// TIA Portal V20 export
FUNCTION_BLOCK "SysPos"   // FB2010, FBD
TITLE = manage a standard positioning system
{ S7_Optimized_Access := 'TRUE' }
AUTHOR : MiCROTEC
VERSION : 1.2
// -2017.03 : Martin
// stored: AutoNumber false, MemoryReserve 100, SetENOAutomatically false
   VAR_INPUT
      actual { ExternalAccessible := 'False'; ExternalVisible := 'False'; ExternalWritable := 'False'} : Real;   // actual position
      target { ExternalAccessible := 'False'; ExternalVisible := 'False'; ExternalWritable := 'False'} : Real;   // target position , start new position only if target position change
      tarMinPos { ExternalAccessible := 'False'; ExternalVisible := 'False'; ExternalWritable := 'False'} : Real;   // target position minimum
      tarMaxPos { ExternalAccessible := 'False'; ExternalVisible := 'False'; ExternalWritable := 'False'} : Real;   // target position maximum
      tolerance { ExternalAccessible := 'False'; ExternalVisible := 'False'; ExternalWritable := 'False'} : Real;   // tolerance for output signal position ok
      regPoint { ExternalAccessible := 'False'; ExternalVisible := 'False'; ExternalWritable := 'False'} : Real;   // regulation point (stop point before target position)
      regOn { ExternalAccessible := 'False'; ExternalVisible := 'False'; ExternalWritable := 'False'} : Bool;   // continuouse regulation on
      restart { ExternalAccessible := 'False'; ExternalVisible := 'False'; ExternalWritable := 'False'} : Bool;   // restart new positioning
      auto { ExternalAccessible := 'False'; ExternalVisible := 'False'; ExternalWritable := 'False'} : Bool;   // automatic (manP/manM and gain works only if auto is on)
      manP { ExternalAccessible := 'False'; ExternalVisible := 'False'; ExternalWritable := 'False'} : Bool;   // manual button plus
      manM { ExternalAccessible := 'False'; ExternalVisible := 'False'; ExternalWritable := 'False'} : Bool;   // manual button minus
      manPValue { ExternalAccessible := 'False'; ExternalVisible := 'False'; ExternalWritable := 'False'} : Real := 10.0;   // increase value in hand mode
      manMValue { ExternalAccessible := 'False'; ExternalVisible := 'False'; ExternalWritable := 'False'} : Real := 10.0;   // decrease value in hand mode
      stopRamp { ExternalAccessible := 'False'; ExternalVisible := 'False'; ExternalWritable := 'False'} : Real;   // position for stopramp
      stopSpeed { ExternalAccessible := 'False'; ExternalVisible := 'False'; ExternalWritable := 'False'} : Real;   // minimum speed for stopramp [0.0-1.0]
      approachPoint { ExternalAccessible := 'False'; ExternalVisible := 'False'; ExternalWritable := 'False'} : Real;   // aproach point, if its 0 than its OFF
   END_VAR
   VAR_OUTPUT
      plus { ExternalAccessible := 'False'; ExternalVisible := 'False'; ExternalWritable := 'False'} : Bool;   // command plus
      minus { ExternalAccessible := 'False'; ExternalVisible := 'False'; ExternalWritable := 'False'} : Bool;   // command minus
      slow { ExternalAccessible := 'False'; ExternalVisible := 'False'; ExternalWritable := 'False'} : Bool;   // slow
      posOk { ExternalAccessible := 'False'; ExternalVisible := 'False'; ExternalWritable := 'False'} : Bool;   // position ok
      tar { ExternalAccessible := 'False'; ExternalVisible := 'False'; ExternalWritable := 'False'} : Real;   // target position
      speedGain { ExternalAccessible := 'False'; ExternalVisible := 'False'; ExternalWritable := 'False'} : Real;   // gain for speed regulation ["StopSpeed" to 1.0]
   END_VAR
   VAR_IN_OUT
      Enc : "TypeEncoder";
   END_VAR
   VAR
      var { ExternalAccessible := 'False'; ExternalVisible := 'False'; ExternalWritable := 'False'} : Struct
         "bool" : Bool;
         "byte" : Byte;
         "word" : Word;
         "dword" : DWord;
         "int" : Int;
         "dint" : DInt;
         "real" : Real;
         s5time : S5Time;
         "time" : Time;
         hm : Array[1..16] of Bool;
         fm : Array[1..16] of Bool;
      END_STRUCT;
      statTargetOld { ExternalAccessible := 'False'; ExternalVisible := 'False'; ExternalWritable := 'False'} : Real;
      statApproachPoint { ExternalAccessible := 'False'; ExternalVisible := 'False'; ExternalWritable := 'False'} : Real;
      statRegPlusPos { ExternalAccessible := 'False'; ExternalVisible := 'False'; ExternalWritable := 'False'} : Real;
      statRegMinusPos { ExternalAccessible := 'False'; ExternalVisible := 'False'; ExternalWritable := 'False'} : Real;
      statInTolerance { ExternalAccessible := 'False'; ExternalVisible := 'False'; ExternalWritable := 'False'} : Bool;
      statAproachRun { ExternalAccessible := 'False'; ExternalVisible := 'False'; ExternalWritable := 'False'} : Bool;
      StatPosOk { ExternalAccessible := 'False'; ExternalVisible := 'False'; ExternalWritable := 'False'} : Bool;
      statSpeedDelta { ExternalAccessible := 'False'; ExternalVisible := 'False'; ExternalWritable := 'False'} : Real;
      statSpeedPerMm { ExternalAccessible := 'False'; ExternalVisible := 'False'; ExternalWritable := 'False'} : Real;
      statTarMin { ExternalAccessible := 'False'; ExternalVisible := 'False'; ExternalWritable := 'False'} : Bool;
      statTarMax { ExternalAccessible := 'False'; ExternalVisible := 'False'; ExternalWritable := 'False'} : Bool;
      statTar { ExternalAccessible := 'False'; ExternalVisible := 'False'; ExternalWritable := 'False'} : Real;
      statPlus { ExternalAccessible := 'False'; ExternalVisible := 'False'; ExternalWritable := 'False'} : Bool;
      statMinus { ExternalAccessible := 'False'; ExternalVisible := 'False'; ExternalWritable := 'False'} : Bool;
      statSpeedGain { ExternalAccessible := 'False'; ExternalVisible := 'False'; ExternalWritable := 'False'} : Real;
      statSlow { ExternalAccessible := 'False'; ExternalVisible := 'False'; ExternalWritable := 'False'} : Bool;
      statTarMaxPosOld : Real;
      statTarMinPosOld : Real;
   END_VAR
   VAR_TEMP   // added for the SCL form of the ladder/FBD networks
      _w1 : Bool;
      _w2 : Bool;
      _w3 : Bool;
   END_VAR
BEGIN

REGION Network 1: manual change target position
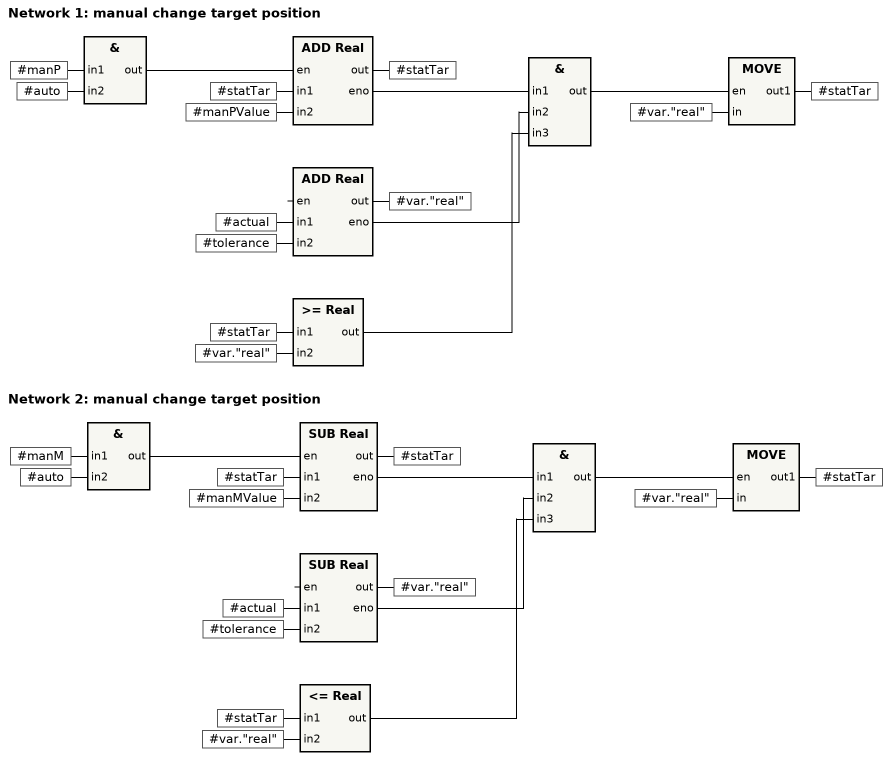
   // ENO of a box is taken as its EN; it also drops when the box reports an error
   #_w1 := #manP AND #auto;
   IF #_w1 THEN #statTar := #statTar + #manPValue; END_IF;
   #var."real" := #actual + #tolerance;
   IF #_w1 AND (#statTar >= #var."real") THEN #statTar := #var."real"; END_IF;
END_REGION

REGION Network 2: manual change target position
   // ENO of a box is taken as its EN; it also drops when the box reports an error
   #_w1 := #manM AND #auto;
   IF #_w1 THEN #statTar := #statTar - #manMValue; END_IF;
   #var."real" := #actual - #tolerance;
   IF #_w1 AND (#statTar <= #var."real") THEN #statTar := #var."real"; END_IF;
END_REGION

REGION Network 3: start positioning
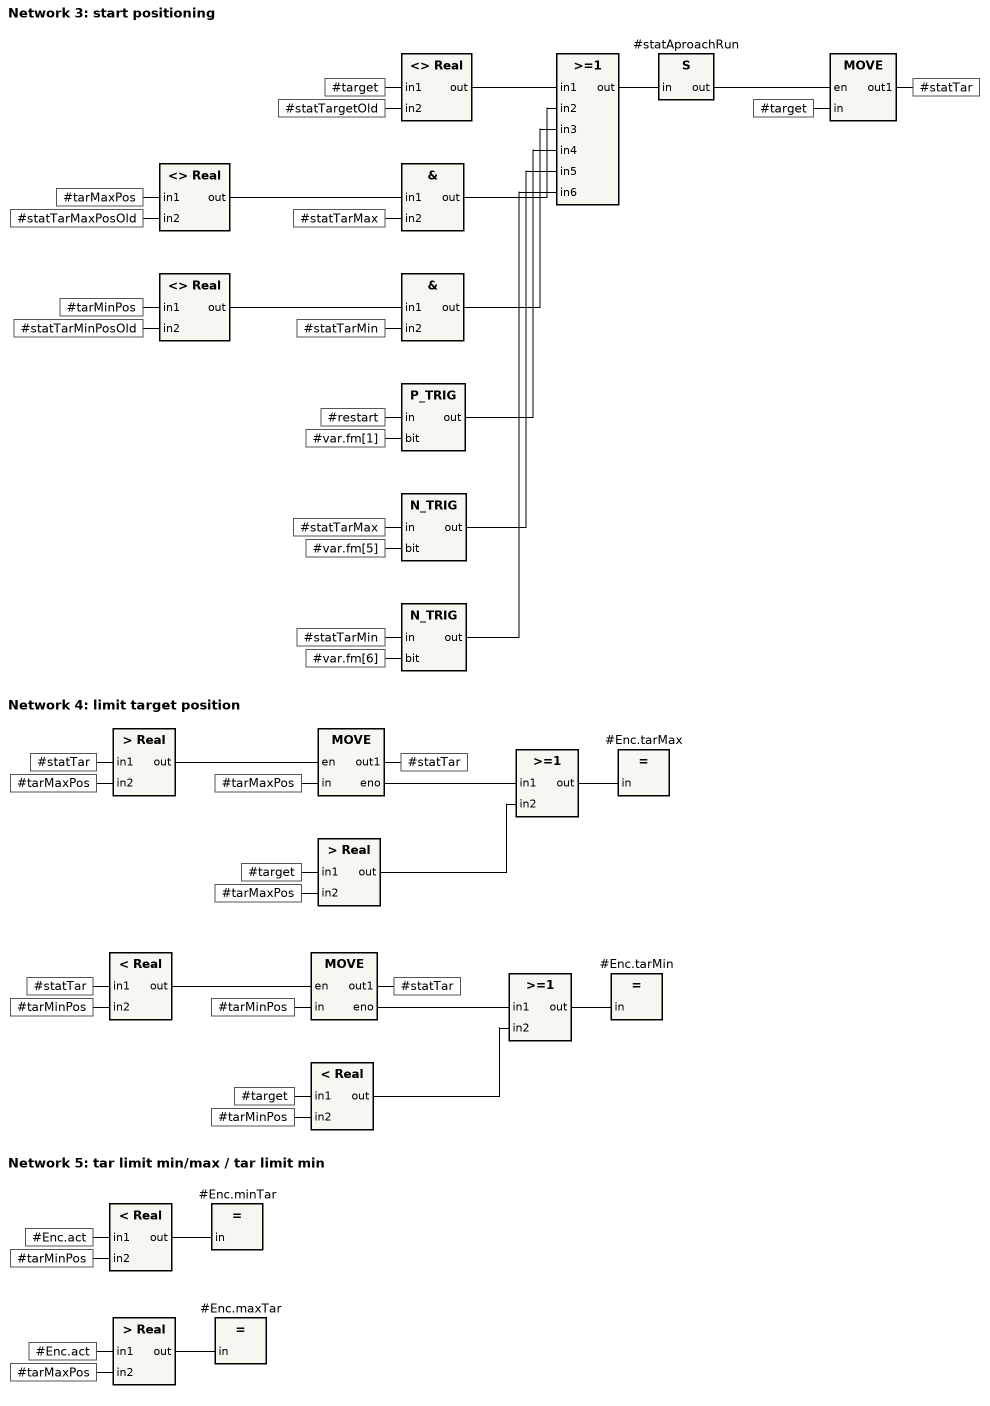
   #_w1 := #restart AND NOT #var.fm[1];   // rising edge
   #var.fm[1] := #restart;
   #_w2 := NOT #statTarMax AND #var.fm[5];   // falling edge
   #var.fm[5] := #statTarMax;
   #_w3 := NOT #statTarMin AND #var.fm[6];   // falling edge
   #var.fm[6] := #statTarMin;
   IF (#target <> #statTargetOld) OR ((#tarMaxPos <> #statTarMaxPosOld) AND #statTarMax) OR ((#tarMinPos <> #statTarMinPosOld) AND #statTarMin) OR #_w1 OR #_w2 OR #_w3 THEN
       #statAproachRun := TRUE;
       #statTar := #target;
   END_IF;
END_REGION

REGION Network 4: limit target position
   // ENO of a box is taken as its EN; it also drops when the box reports an error
   #_w1 := #statTar > #tarMaxPos;
   IF #_w1 THEN #statTar := #tarMaxPos; END_IF;
   #Enc.tarMax := #_w1 OR (#target > #tarMaxPos);
   #_w2 := #statTar < #tarMinPos;
   IF #_w2 THEN #statTar := #tarMinPos; END_IF;
   #Enc.tarMin := #_w2 OR (#target < #tarMinPos);
END_REGION

REGION Network 5: tar limit min/max / tar limit min
   #Enc.minTar := #Enc.act < #tarMinPos;
   #Enc.maxTar := #Enc.act > #tarMaxPos;
END_REGION

REGION Network 6 (SCL): approach/regulation point
   #statApproachPoint := #statTar + #approachPoint;

   #statRegMinusPos := #statTar - #regPoint;
   #statRegPlusPos := #statTar + #regPoint;
END_REGION

REGION Network 7: approachpoint reach
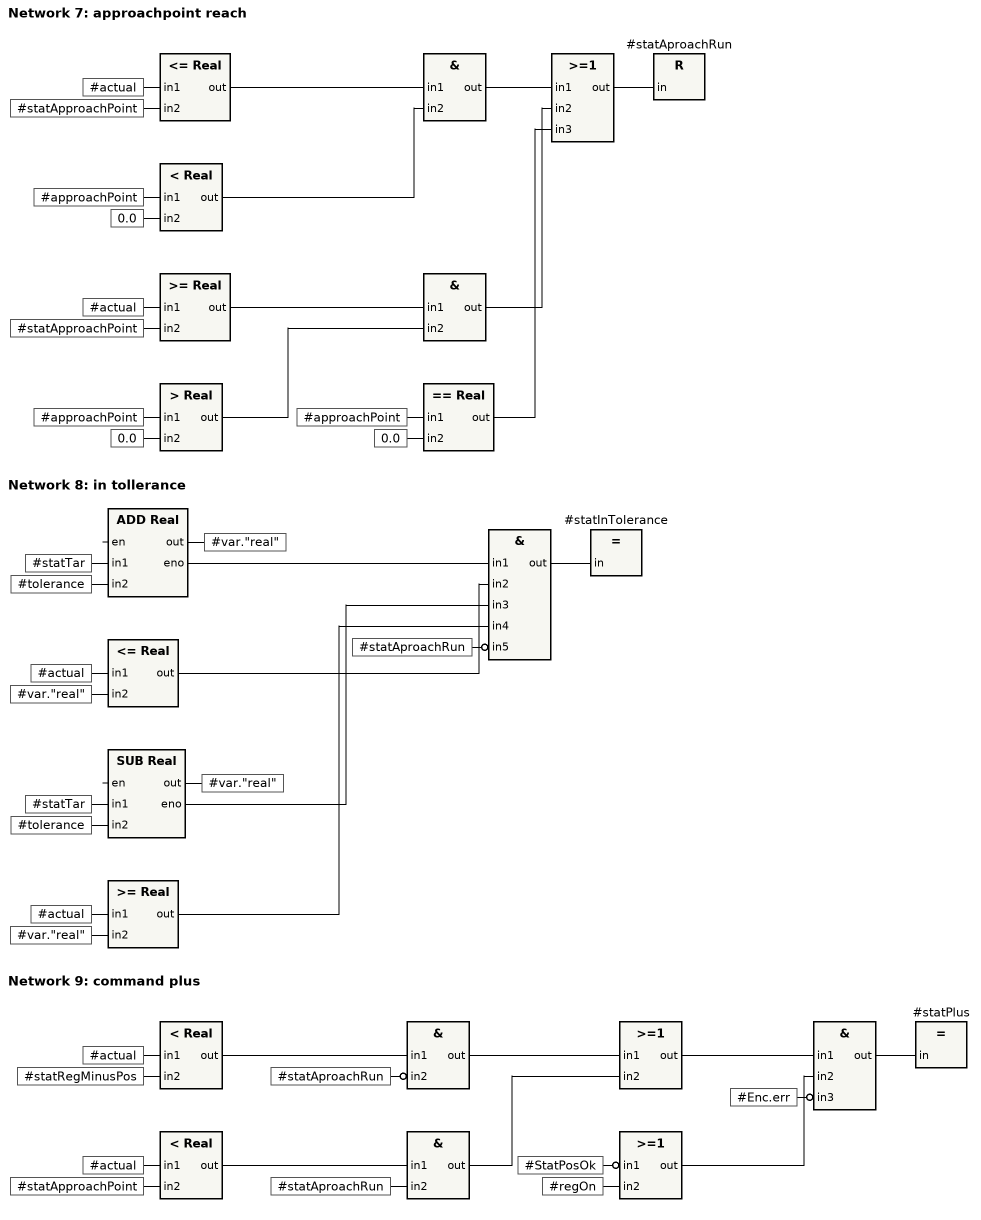
   IF ((#actual <= #statApproachPoint) AND (#approachPoint < 0.0)) OR ((#actual >= #statApproachPoint) AND (#approachPoint > 0.0)) OR (#approachPoint = 0.0) THEN
       #statAproachRun := FALSE;
   END_IF;
END_REGION

REGION Network 8: in tollerance
   // ENO of a box is taken as its EN; it also drops when the box reports an error
   #var."real" := #statTar + #tolerance;
   #_w1 := #actual <= #var."real";
   #var."real" := #statTar - #tolerance;
   #statInTolerance := #_w1 AND (#actual >= #var."real") AND NOT #statAproachRun;
END_REGION

REGION Network 9: command plus
   #statPlus := (((#actual < #statRegMinusPos) AND NOT #statAproachRun) OR ((#actual < #statApproachPoint) AND #statAproachRun)) AND (NOT #StatPosOk OR #regOn) AND NOT #Enc.err;
END_REGION

REGION Network 10: command minus
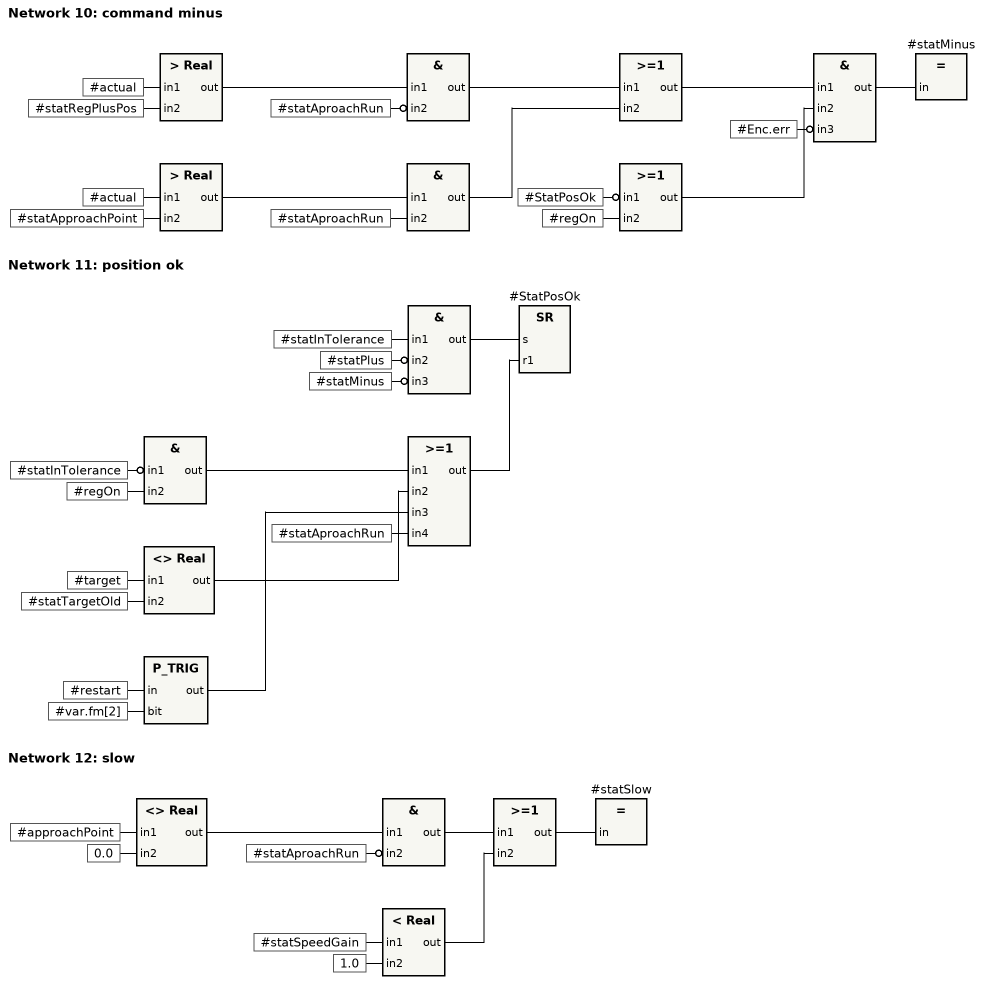
   #statMinus := (((#actual > #statRegPlusPos) AND NOT #statAproachRun) OR ((#actual > #statApproachPoint) AND #statAproachRun)) AND (NOT #StatPosOk OR #regOn) AND NOT #Enc.err;
END_REGION

REGION Network 11: position ok
   #_w1 := #restart AND NOT #var.fm[2];   // rising edge
   #var.fm[2] := #restart;
   IF #statInTolerance AND NOT #statPlus AND NOT #statMinus THEN
       #StatPosOk := TRUE;   // SR flip-flop
   END_IF;
   IF (NOT #statInTolerance AND #regOn) OR (#target <> #statTargetOld) OR #_w1 OR #statAproachRun THEN
       #StatPosOk := FALSE;
   END_IF;
END_REGION

REGION Network 12: slow
   #statSlow := ((#approachPoint <> 0.0) AND NOT #statAproachRun) OR (#statSpeedGain < 1.0);
END_REGION

REGION Network 13 (SCL): old position
   #statTargetOld := #target;
   #statTarMaxPosOld := #tarMaxPos;
   #statTarMinPosOld := #tarMinPos;
END_REGION

REGION Network 14 (SCL): speed gain for stop ramp
   #statSpeedDelta := 1.0 - #stopSpeed;
   #statSpeedPerMm := #statSpeedDelta / #stopRamp;
   #statSpeedGain := #stopSpeed + ABS_REAL((#statTar - #actual) * #statSpeedPerMm);

   IF #statSpeedGain < #stopSpeed THEN
       #statSpeedGain := #stopSpeed;
   END_IF;

   IF #statSpeedGain > 1.0 OR NOT #auto THEN
       #statSpeedGain := 1.0;
   END_IF;
END_REGION

REGION Network 15 (SCL): write outputs
       #plus := #statPlus;
       #minus := #statMinus;
       #slow:= #statSlow;
       #posOk := #StatPosOk;
       #tar := #statTar;
       #speedGain := #statSpeedGain;
END_REGION

REGION Network 16 (SCL): in/out data
       #Enc.tarMinPos := #tarMinPos;
       #Enc.tarMaxPos := #tarMaxPos;
       #Enc.act := #actual;
       #Enc.tar := #statTar;
       #Enc.posOk := #StatPosOk;
END_REGION
END_FUNCTION_BLOCK
